Staubli VAL3: getSizeItem.pgx

public program getSizeItem(num& x_nSize[])
begin
  // get the size
  if pEdit.iEvent.sType==""
    x_nSize=0
  else
    x_nSize=size(pEdit.iEvent)
  endIf
end
